Staubli VAL3: remTransIP.pgx

program remTransIP(string& sArgs[] (dimensions=1), string& sReturn[] (dimensions=1))
  local bool bOk
  local num nLoop
  local num nVal
  local string sArgsLoop
  local trsf trUser
begin
  //Translates the current interaction point.
  //
  logMsg("call remTransIP")
  trUser={0,0,0,0,0,0}
  nLoop=0
  sArgsLoop=sArgs
  while nLoop<3
    sArgsLoop=toNum(sArgsLoop,nVal,bOk)
    if bOk
      switch nLoop
        case 0
          trUser.x=nVal
        break
        case 1
          trUser.y=nVal
        break
        case 2
          trUser.z=nVal
        break
      endSwitch
      nLoop=nLoop+1
    else
      call remErrNum("CMDTRANSIP",sArgs,sReturn)
      return
    endIf
  endWhile
  if nIPNumber==0
    fIP1.trsf=fIP1.trsf*trUser
  else
    fIP2.trsf=fIP2.trsf*trUser
  endIf
  sReturn="CMDTRANSIP"
end
